# EPICS autosave request: DRIVERNAMELOWERSHORTApp/Db/ADDRIVERNAMESTANDARD_settings.req
file "ADBase_settings.req", P=$(P),  R=image1:
